TYPE TerminalStatus :
STRUCT
    WorkingCounterError : BOOL;
    IOError : BOOL;
END_STRUCT
END_TYPE

(* stored: Version 1.1.0.1, ProductVersion 3.1.4024.4
   DUT TerminalStatus: Id {08ca8f15-33b5-40ce-a262-dcd3398b9cfb} *)
